FUNCTION DWORDS_TO_ARR08B (* this Function combines 2 DWORDSs to a 8-BYTE Array; Little-Endian-Format (Intel-Standard) *)
  (* Standard: 61499-1; Description: Copyright (c) 2024 HR Agrartechnik GmbH This program and the accompanying materials are made available under the terms of the Eclipse Public License 2.0 which is available at https://www.eclipse.org/legal/epl-2.0/ SPDX-License-Identifier: EPL-2.0 Little-Endian-Format (Intel-Standard) PC-basierte Steuerungen (Beckhoff, Wago, B&R, Raspberry Pi) *)
  (* Version 1.0, 2024-02-22, Franz Höpfinger, HR Agrartechnik GmbH *)
  PACKAGE logiBUS::utils::conversion::arr::reversing;
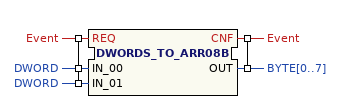
  EVENT_INPUT
    REQ WITH IN_00, IN_01;
  END_EVENT
  EVENT_OUTPUT
    CNF WITH OUT;
  END_EVENT
  VAR_INPUT
    IN_00 : DWORD; (* DWORD 00 *)
    IN_01 : DWORD; (* DWORD 01 *)
  END_VAR
  VAR_OUTPUT
    OUT : ARRAY [0..7] OF BYTE; (* ARR08B Output *)
  END_VAR
  BODY IN ST:
PACKAGE logiBUS::utils::conversion::arr::reversing;

(* this Function combines 2 DWORDSs to a 8-BYTE Array; Little-Endian-Format (Intel-Standard) *)
FUNCTION DWORDS_TO_ARR08B

VAR_INPUT
	IN_00 : DWORD; // DWORD 00
	IN_01 : DWORD; // DWORD 01
END_VAR

VAR_OUTPUT
	OUT : ARRAY[0..7] OF BYTE; // ARR08B Output
END_VAR

OUT[0] := IN_00.%B0;
OUT[1] := IN_00.%B1;
OUT[2] := IN_00.%B2;
OUT[3] := IN_00.%B3;
OUT[4] := IN_01.%B0;
OUT[5] := IN_01.%B1;
OUT[6] := IN_01.%B2;
OUT[7] := IN_01.%B3;

END_FUNCTION
  END_BODY
END_FUNCTION
